// TIA Portal V18 export
TYPE "UDT_DIbasic"
// stored: IsFailsafeCompliant false
   STRUCT
      iID : DInt;   // DIs ID for monitoring
      iCounter : Int;   // Counter for DIs EDGE
      xFiltered : Bool;   // Filtered value
      wMark : String["IOmark_string_length"];   // DIs label for monitoring
      iAddImpOff : Int;   // Temp
      iAddImpOn : Int;   // Temp
      xMemory : Bool;   // Temp
   END_STRUCT;
END_TYPE
